// TIA Portal V16 export
// export: Created 2023-03-29T11:05:04.6808886Z, ExportSetting WithDefaults, DisplayName Totally Integrated Automation Portal, DisplayVersion V16 Update 6, DisplayName TIA Portal Version Control Interface, DisplayVersion V16 Update 2, DisplayName TIA Portal Openness, DisplayVersion V16 Update 6, DisplayName STEP 7 Professional, DisplayVersion V16 Update 6, DisplayName STEP 7 Safety, DisplayVersion V16, DisplayName WinCC Advanced, DisplayVersion V16 Update 6
VAR_GLOBAL   // PLC tag table "tags"
   "Tuning.TIR_visible" AT %M1002.0 : Bool;
   "Tuning.SUT_visible" AT %M1002.1 : Bool;
   "Tuning.Mode_visible" AT %M1002.2 : Bool;
   "PID_Compact.State" AT %MW1004 : Int;
   "PID_Compact.Setpoint" AT %MD1006 : Real;
   "PID_Compact.ScaledInput" AT %MD1010 : Real;
   "PID_Compact.Output_PWM" AT %M1014.0 : Bool;
   "PID_Compact.ModeActivate" AT %M1014.1 : Bool;
   "PID_Compact.ManualEnable" AT %M1014.2 : Bool;
   "PID_Compact.Disturbance" AT %MD1016 : Real;
   "HMI.Setpoint_limited" AT %M1020.0 : Bool;
   "HMI.PhysicalUnit" AT %MB1021 : Char;
   "HMI.Output_PWM_USInt" AT %MB1022 : USInt;
   "HMI.ManualMode_visible(1)" AT %M1023.0 : Bool;
   "HMI.ManualMode_visible" AT %M1023.1 : Bool;
   "HMI.ErrorBits_Int" AT %MW1024 : Int;
   "HMI.ErrorAck_Int" AT %MW1026 : Int;
   "HMI.Warning_Int" AT %MW1028 : Int;
   "HMI.ErrorAck" AT %M1030.0 : Bool;
   "HMI.Acknowledge_visible" AT %M1030.1 : Bool;
   Communication_Alarm AT %M1030.2 : Bool;   // Znacznik błedu komunikacji HMI - PLC
   outAlarm AT %M1030.3 : Bool;   // Znacznik alarmu zbiorczego (Sygnalizator)
   "HMI.alarm_byte_1" AT %MW800 : Word;   // słowo alarmów
   "HMI.gotowość_falownik_1" AT %M800.0 : Bool;   // gotowość falownika 1
   "HMI.brak_zasilania" AT %M800.1 : Bool;   // brak zasilnia
   "HMI.SłowoStatus_Falownik1" AT %MW2000 : Int;   // Słowo statusu falownika F1
   "HMI.FalSata_bit_0" AT %M2000.0 : Bool;   // Sterowanie poprawne
   "HMI.FalSata_bit_1" AT %M2000.1 : Bool;   // falownik gotowość
   "HMI.FalSata_bit_2" AT %M2000.2 : Bool;   // wybieg
   "HMI.FalSata_bit_3" AT %M2000.3 : Bool;   // trip error
   "HMI.FalSata_bit_4" AT %M2000.4 : Bool;   // no trip error
   "HMI.FalSata_bit_5" AT %M2000.5 : Bool;   // reserved
   "HMI.FalSata_bit_6" AT %M2000.6 : Bool;   // trip zablokowany
   "HMI.FalSata_bit_7" AT %M2000.7 : Bool;   // Ostrzeżenie
   "HMI.FalSata_bit_8" AT %M2001.0 : Bool;   // prędkość = referencyjnej
   "HMI.FalSata_bit_9" AT %M2001.1 : Bool;   // listwa sterowania
   "HMI.FalSata_bit_10" AT %M2001.2 : Bool;   // częstotliwość ok
   "HMI.FalSata_bit_11" AT %M2001.3 : Bool;   // praca
   "HMI.FalSata_bit_12" AT %M2001.4 : Bool;   // rezystor hamowania
   "HMI.FalSata_bit_13" AT %M2001.5 : Bool;   // volty przekroczone
   "HMI.FalSata_bit_14" AT %M2001.6 : Bool;   // problem z momentem obrotowym
   "HMI.FalSata_bit_15" AT %M2001.7 : Bool;   // zabezpieczenie termiczne
   "HMI.kasowanie.ekranów" AT %MW1000 : Int;
   "HMI.kasowanie.ekranów_bit_0" AT %M1000.0 : Bool;   // kasowanie alarmu ekran pomp
   "HMI.kasowanie.ekranów_bit_1" AT %M1000.1 : Bool;   // kasowanie alarmu ekran zasów
   "HMI.kasowanie.ekranów_bit_2" AT %M1000.2 : Bool;
   "HMI.kasowanie.ekranów_bit_3" AT %M1000.3 : Bool;
   "HMI.kasowanie.ekranów_bit_4" AT %M1000.4 : Bool;
   "HMI.kasowanie.ekranów_bit_5" AT %M1000.5 : Bool;
   "HMI.kasowanie.ekranów_bit_6" AT %M1000.6 : Bool;
   "HMI.kasowanie.ekranów_bit_7" AT %M1000.7 : Bool;
   "HMI.alarm_01" AT %M1001.0 : Bool;   // Alarm Modbus RTU
   "HMI.alarm_02" AT %M1001.1 : Bool;   // Ostrzerzenie Modbus RTU
   "HMI.alarm_01(2)" AT %M1001.2 : Bool;
   "HMI.alarm_01(3)" AT %M1001.3 : Bool;
   "HMI.alarm_01(4)" AT %M1001.4 : Bool;
   "HMI.alarm_01(5)" AT %M1001.5 : Bool;
   "HMI.alarm_01(6)" AT %M1001.6 : Bool;
   "HMI.alarm_01(7)" AT %M1001.7 : Bool;
END_VAR
